% RSLogix 500 project PV10.RSS, saved by version 8.30.00.16 %
PROJECT "PV10"    % processor: Bul.1763 MicroLogix 1100 Series B %

PROGRAM FILES
  LAD 2   44 rungs

DATA FILES
  O0 OUTPUT  5 elements
  I1 INPUT  7 elements
  S2 STATUS  66 elements
  B3 BINARY  4 elements
  T4 TIMER  5 elements
  C5 COUNTER  2 elements
  R6 CONTROL  1 elements
  N7 INTEGER  3 elements
  F8 FLOAT  1 elements

LADDER 2
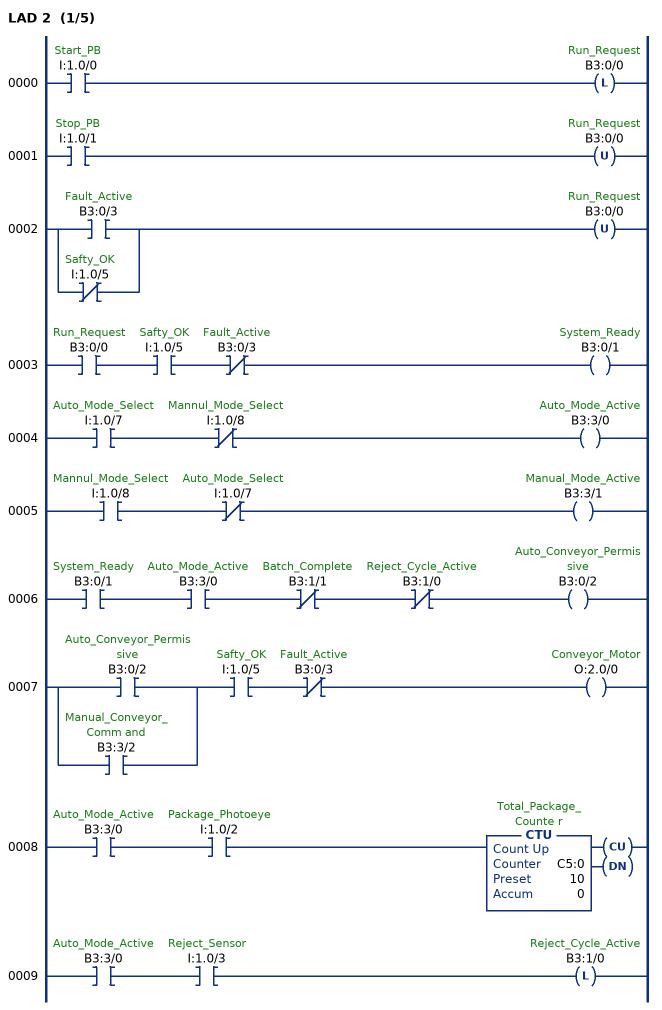
% Rung: 0 %
SOR XIC I:1.0/0 OTL B3:0/0 EOR
%   I:1.0/0  "Start_PB" %
%   B3:0/0  "Run_Request" %
% Rung: 1 %
SOR XIC I:1.0/1 OTU B3:0/0 EOR
%   I:1.0/1  "Stop_PB" %
%   B3:0/0  "Run_Request" %
% Rung: 2 %
SOR BST XIC B3:0/3 NXB XIO I:1.0/5 BND OTU B3:0/0 EOR
%   B3:0/3  "Fault_Active" %
%   I:1.0/5  "Safty_OK" %
%   B3:0/0  "Run_Request" %
% Rung: 3 %
SOR XIC B3:0/0 XIC I:1.0/5 XIO B3:0/3 OTE B3:0/1 EOR
%   B3:0/0  "Run_Request" %
%   I:1.0/5  "Safty_OK" %
%   B3:0/3  "Fault_Active" %
%   B3:0/1  "System_Ready" %
% Rung: 4 %
SOR XIC I:1.0/7 XIO I:1.0/8 OTE B3:3/0 EOR
%   I:1.0/7  "Auto_Mode_Select" %
%   I:1.0/8  "Mannul_Mode_Select" %
%   B3:3/0  "Auto_Mode_Active" %
% Rung: 5 %
SOR XIC I:1.0/8 XIO I:1.0/7 OTE B3:3/1 EOR
%   I:1.0/8  "Mannul_Mode_Select" %
%   I:1.0/7  "Auto_Mode_Select" %
%   B3:3/1  "Manual_Mode_Active" %
% Rung: 6 %
SOR XIC B3:0/1 XIC B3:3/0 XIO B3:1/1 XIO B3:1/0 OTE B3:0/2 EOR
%   B3:0/1  "System_Ready" %
%   B3:3/0  "Auto_Mode_Active" %
%   B3:1/1  "Batch_Complete" %
%   B3:1/0  "Reject_Cycle_Active" %
%   B3:0/2  "Auto_Conveyor_Permis sive" %
% Rung: 7 %
SOR BST XIC B3:0/2 NXB XIC B3:3/2 BND XIC I:1.0/5 XIO B3:0/3 OTE O:2.0/0 EOR
%   B3:0/2  "Auto_Conveyor_Permis sive" %
%   B3:3/2  "Manual_Conveyor_Comm and" %
%   I:1.0/5  "Safty_OK" %
%   B3:0/3  "Fault_Active" %
%   O:2.0/0  "Conveyor_Motor" %
% Rung: 8 %
SOR XIC B3:3/0 XIC I:1.0/2 CTU C5:0 10 0 EOR
%   B3:3/0  "Auto_Mode_Active" %
%   I:1.0/2  "Package_Photoeye" %
%   C5:0  "Total_Package_Counte r" %
% Rung: 9 %
SOR XIC B3:3/0 XIC I:1.0/3 OTL B3:1/0 EOR
%   B3:3/0  "Auto_Mode_Active" %
%   I:1.0/3  "Reject_Sensor" %
%   B3:1/0  "Reject_Cycle_Active" %

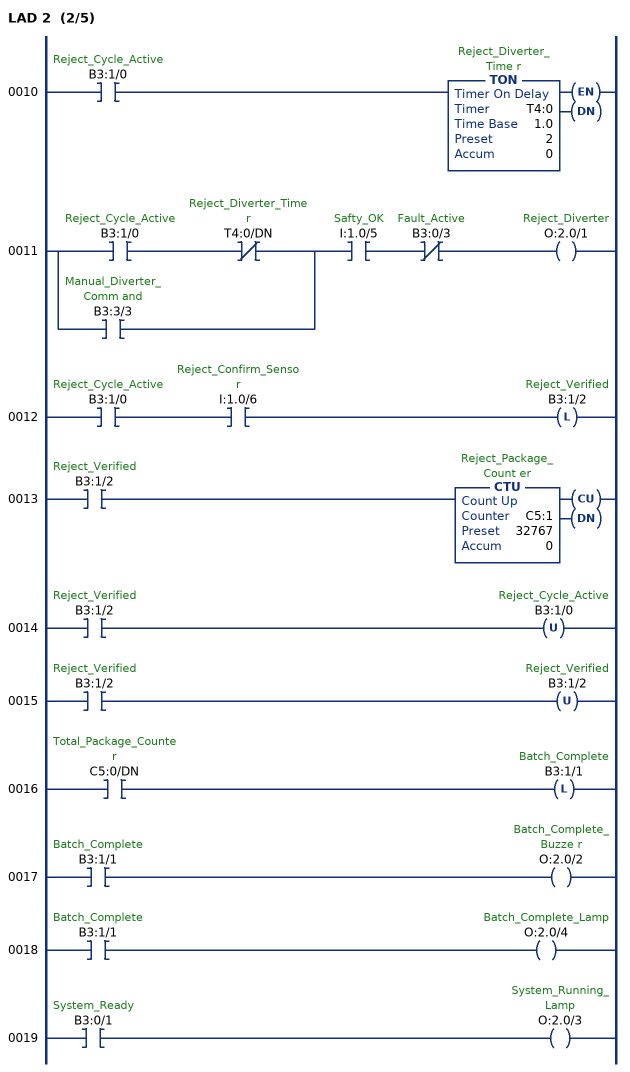
% Rung: 10 %
SOR XIC B3:1/0 TON T4:0 1.0 2 0 EOR
%   B3:1/0  "Reject_Cycle_Active" %
%   T4:0  "Reject_Diverter_Time r" %
% Rung: 11 %
SOR BST XIC B3:1/0 XIO T4:0/DN NXB XIC B3:3/3 BND XIC I:1.0/5 XIO B3:0/3 OTE O:2.0/1 EOR
%   B3:1/0  "Reject_Cycle_Active" %
%   T4:0  "Reject_Diverter_Time r" %
%   B3:3/3  "Manual_Diverter_Comm and" %
%   I:1.0/5  "Safty_OK" %
%   B3:0/3  "Fault_Active" %
%   O:2.0/1  "Reject_Diverter" %
% Rung: 12 %
SOR XIC B3:1/0 XIC I:1.0/6 OTL B3:1/2 EOR
%   B3:1/0  "Reject_Cycle_Active" %
%   I:1.0/6  "Reject_Confirm_Senso r" %
%   B3:1/2  "Reject_Verified" %
% Rung: 13 %
SOR XIC B3:1/2 CTU C5:1 32767 0 EOR
%   B3:1/2  "Reject_Verified" %
%   C5:1  "Reject_Package_Count er" %
% Rung: 14 %
SOR XIC B3:1/2 OTU B3:1/0 EOR
%   B3:1/2  "Reject_Verified" %
%   B3:1/0  "Reject_Cycle_Active" %
% Rung: 15 %
SOR XIC B3:1/2 OTU B3:1/2 EOR
%   B3:1/2  "Reject_Verified" %
% Rung: 16 %
SOR XIC C5:0/DN OTL B3:1/1 EOR
%   C5:0  "Total_Package_Counte r" %
%   B3:1/1  "Batch_Complete" %
% Rung: 17 %
SOR XIC B3:1/1 OTE O:2.0/2 EOR
%   B3:1/1  "Batch_Complete" %
%   O:2.0/2  "Batch_Complete_Buzze r" %
% Rung: 18 %
SOR XIC B3:1/1 OTE O:2.0/4 EOR
%   B3:1/1  "Batch_Complete" %
%   O:2.0/4  "Batch_Complete_Lamp" %
% Rung: 19 %
SOR XIC B3:0/1 OTE O:2.0/3 EOR
%   B3:0/1  "System_Ready" %
%   O:2.0/3  "System_Running_Lamp" %

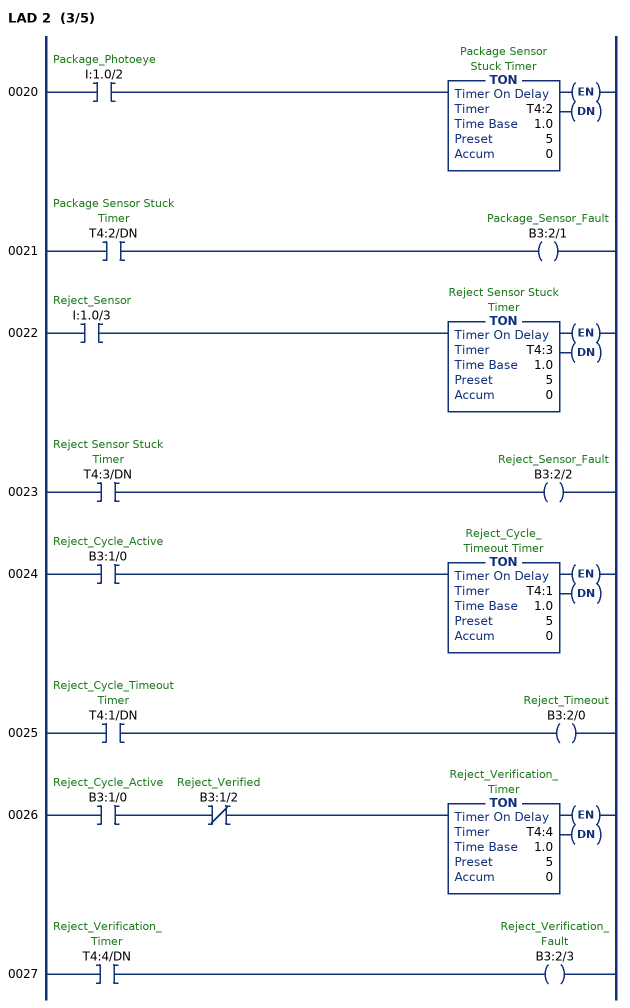
% Rung: 20 %
SOR XIC I:1.0/2 TON T4:2 1.0 5 0 EOR
%   I:1.0/2  "Package_Photoeye" %
%   T4:2  "Package Sensor Stuck Timer" %
% Rung: 21 %
SOR XIC T4:2/DN OTE B3:2/1 EOR
%   T4:2  "Package Sensor Stuck Timer" %
%   B3:2/1  "Package_Sensor_Fault" %
% Rung: 22 %
SOR XIC I:1.0/3 TON T4:3 1.0 5 0 EOR
%   I:1.0/3  "Reject_Sensor" %
%   T4:3  "Reject Sensor Stuck Timer" %
% Rung: 23 %
SOR XIC T4:3/DN OTE B3:2/2 EOR
%   T4:3  "Reject Sensor Stuck Timer" %
%   B3:2/2  "Reject_Sensor_Fault" %
% Rung: 24 %
SOR XIC B3:1/0 TON T4:1 1.0 5 0 EOR
%   B3:1/0  "Reject_Cycle_Active" %
%   T4:1  "Reject_Cycle_Timeout Timer" %
% Rung: 25 %
SOR XIC T4:1/DN OTE B3:2/0 EOR
%   T4:1  "Reject_Cycle_Timeout Timer" %
%   B3:2/0  "Reject_Timeout" %
% Rung: 26 %
SOR XIC B3:1/0 XIO B3:1/2 TON T4:4 1.0 5 0 EOR
%   B3:1/0  "Reject_Cycle_Active" %
%   B3:1/2  "Reject_Verified" %
%   T4:4  "Reject_Verification_ Timer" %
% Rung: 27 %
SOR XIC T4:4/DN OTE B3:2/3 EOR
%   T4:4  "Reject_Verification_ Timer" %
%   B3:2/3  "Reject_Verification_ Fault" %

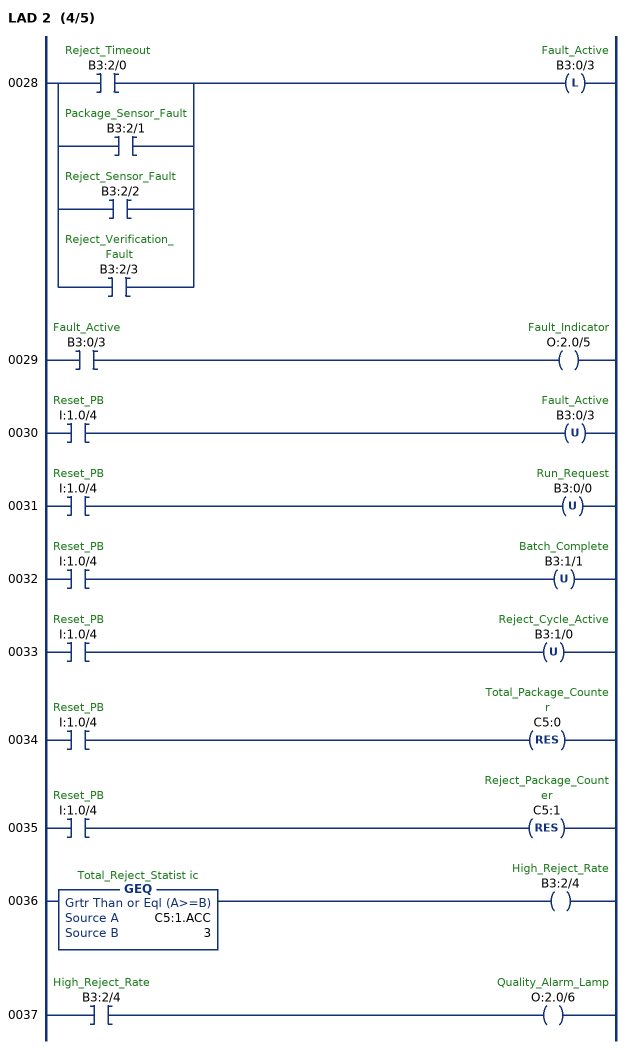
% Rung: 28 %
SOR BST XIC B3:2/0 NXB BST XIC B3:2/1 NXB BST XIC B3:2/2 NXB XIC B3:2/3 BND BND BND OTL B3:0/3 EOR
%   B3:2/0  "Reject_Timeout" %
%   B3:2/1  "Package_Sensor_Fault" %
%   B3:2/2  "Reject_Sensor_Fault" %
%   B3:2/3  "Reject_Verification_ Fault" %
%   B3:0/3  "Fault_Active" %
% Rung: 29 %
SOR XIC B3:0/3 OTE O:2.0/5 EOR
%   B3:0/3  "Fault_Active" %
%   O:2.0/5  "Fault_Indicator" %
% Rung: 30 %
SOR XIC I:1.0/4 OTU B3:0/3 EOR
%   I:1.0/4  "Reset_PB" %
%   B3:0/3  "Fault_Active" %
% Rung: 31 %
SOR XIC I:1.0/4 OTU B3:0/0 EOR
%   I:1.0/4  "Reset_PB" %
%   B3:0/0  "Run_Request" %
% Rung: 32 %
SOR XIC I:1.0/4 OTU B3:1/1 EOR
%   I:1.0/4  "Reset_PB" %
%   B3:1/1  "Batch_Complete" %
% Rung: 33 %
SOR XIC I:1.0/4 OTU B3:1/0 EOR
%   I:1.0/4  "Reset_PB" %
%   B3:1/0  "Reject_Cycle_Active" %
% Rung: 34 %
SOR XIC I:1.0/4 RES C5:0 EOR
%   I:1.0/4  "Reset_PB" %
%   C5:0  "Total_Package_Counte r" %
% Rung: 35 %
SOR XIC I:1.0/4 RES C5:1 EOR
%   I:1.0/4  "Reset_PB" %
%   C5:1  "Reject_Package_Count er" %
% Rung: 36 %
SOR GEQ C5:1.ACC 3 OTE B3:2/4 EOR
%   C5:1.ACC  "Total_Reject_Statist ic" %
%   B3:2/4  "High_Reject_Rate" %
% Rung: 37 %
SOR XIC B3:2/4 OTE O:2.0/6 EOR
%   B3:2/4  "High_Reject_Rate" %
%   O:2.0/6  "Quality_Alarm_Lamp" %

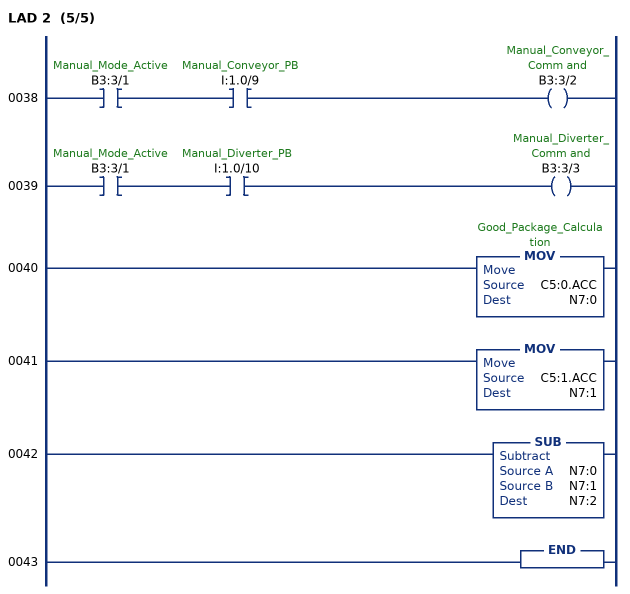
% Rung: 38 %
SOR XIC B3:3/1 XIC I:1.0/9 OTE B3:3/2 EOR
%   B3:3/1  "Manual_Mode_Active" %
%   I:1.0/9  "Manual_Conveyor_PB" %
%   B3:3/2  "Manual_Conveyor_Comm and" %
% Rung: 39 %
SOR XIC B3:3/1 XIC I:1.0/10 OTE B3:3/3 EOR
%   B3:3/1  "Manual_Mode_Active" %
%   I:1.0/10  "Manual_Diverter_PB" %
%   B3:3/3  "Manual_Diverter_Comm and" %
% Rung: 40 %
SOR MOV C5:0.ACC N7:0 EOR
%   C5:0.ACC  "Total_Package_Statis tic" %
%   N7:0  "Good_Package_Calcula tion" %
% Rung: 41 %
SOR MOV C5:1.ACC N7:1 EOR
%   C5:1.ACC  "Total_Reject_Statist ic" %
% Rung: 42 %
SOR SUB N7:0 N7:1 N7:2 EOR
%   N7:0  "Good_Package_Calcula tion" %
% Rung: 43 %
SOR END EOR

DATA TABLE (non-zero values as saved)
DATA B3
% B3:0 % 0X0003 0X0000 0X0000 0X000E
DATA T4
% .PRE .ACC %
% T4:0 % 2 0
% T4:1 % 5 0
% T4:2 % 5 0
% T4:3 % 5 0
% T4:4 % 5 0
DATA C5
% .PRE .ACC %
% C5:0 % 10 0
% C5:1 % 32767 0
